FUNCTION_BLOCK AUI_CTD (* Event driven down counter (Adapter Version) - On Change Triggering *)
  (* Standard: 61499-2; Description: Copyright (c) 2024 HR Agrartechnik GmbH This program and the accompanying materials are made available under the terms of the Eclipse Public License 2.0 which is available at https://www.eclipse.org/legal/epl-2.0/ SPDX-License-Identifier: EPL-2.0 *)
  (* Version 1.0, 2026-04-19, Franz Höpfinger, HR Agrartechnik GmbH, initial API and implementation based on E_CTD with adapter support *)
  PACKAGE adapter::events::unidirectional;
  IMPORT eclipse4diac::core::TypeHash;
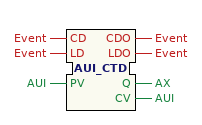
  EVENT_INPUT
    CD; (* Count Down *)
    LD; (* Load CV with PV *)
  END_EVENT
  EVENT_OUTPUT
    CDO; (* Count Down Output *)
    LDO; (* Load Output *)
  END_EVENT
  SOCKETS
    PV : adapter::types::unidirectional::AUI; (* Preset Value *)
  END_SOCKETS
  PLUGS
    Q : adapter::types::unidirectional::AX; (* True if CV <= 0 *)
    CV : adapter::types::unidirectional::AUI; (* Counter Value *)
  END_PLUGS
  VAR
    Q_OLD : BOOL := FALSE; (* Stores the previous state of the output Q to detect changes (On-Change triggering) *) {SET_ATTRIBUTE(Retain, NON_RETAIN)}
  END_VAR
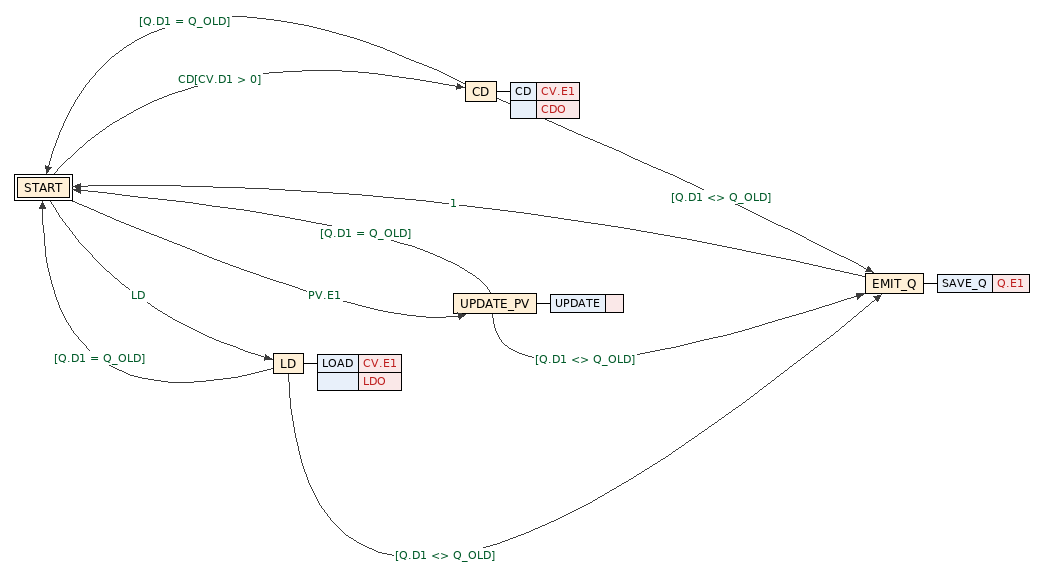
  EC_STATES
    START; (* Initial State *)
    CD : CD -> CV.E1, -> CDO; (* Count Down *)
    LD : LOAD -> CV.E1, -> LDO; (* Load *)
    UPDATE_PV : UPDATE; (* Re-evaluate Q on PV change *)
    EMIT_Q : SAVE_Q -> Q.E1; (* Fires Q event and saves state *)
  END_STATES
  EC_TRANSITIONS
    START TO CD := CD[CV.D1 > 0];
    CD TO EMIT_Q := [Q.D1 <> Q_OLD];
    CD TO START := [Q.D1 = Q_OLD];
    START TO LD := LD;
    LD TO EMIT_Q := [Q.D1 <> Q_OLD];
    LD TO START := [Q.D1 = Q_OLD];
    START TO UPDATE_PV := PV.E1;
    UPDATE_PV TO EMIT_Q := [Q.D1 <> Q_OLD];
    UPDATE_PV TO START := [Q.D1 = Q_OLD];
    EMIT_Q TO START := 1;
  END_TRANSITIONS
  ALGORITHM LOAD IN ST: (* load counter *)
CV.D1 := PV.D1;
Q.D1 := (CV.D1 <= 0);
  END_ALGORITHM
  ALGORITHM CD IN ST: (* count down *)
CV.D1 := CV.D1 - 1;
Q.D1 := (CV.D1 <= 0);
  END_ALGORITHM
  ALGORITHM UPDATE IN ST: (* update status only *)
Q.D1 := (CV.D1 <= 0);
  END_ALGORITHM
  ALGORITHM SAVE_Q IN ST: (* save state *)
Q_OLD := Q.D1;
  END_ALGORITHM
END_FUNCTION_BLOCK
